(* PLC project Unnamed, Unknown Unnamed 1 *)
(* stored: creationDateTime 2023-05-15T12:31:37, modificationDateTime 2023-06-23T13:12:46 *)

PROGRAM thermal_level_controller
  VAR
    in_valve AT %QX0.0 : BOOL := false;
    out_valve AT %QX0.1 : BOOL := false;
    start_button AT %IX0.0 : BOOL := false;
    low_level AT %IX0.1 : BOOL := false;
    high_level AT %IX0.2 : BOOL := false;
    heater_current AT %QW0 : UINT := 0;
    temperature AT %IW0 : UINT := 0;
  END_VAR
  VAR
    thermal_control_active : BOOL := false;
  END_VAR

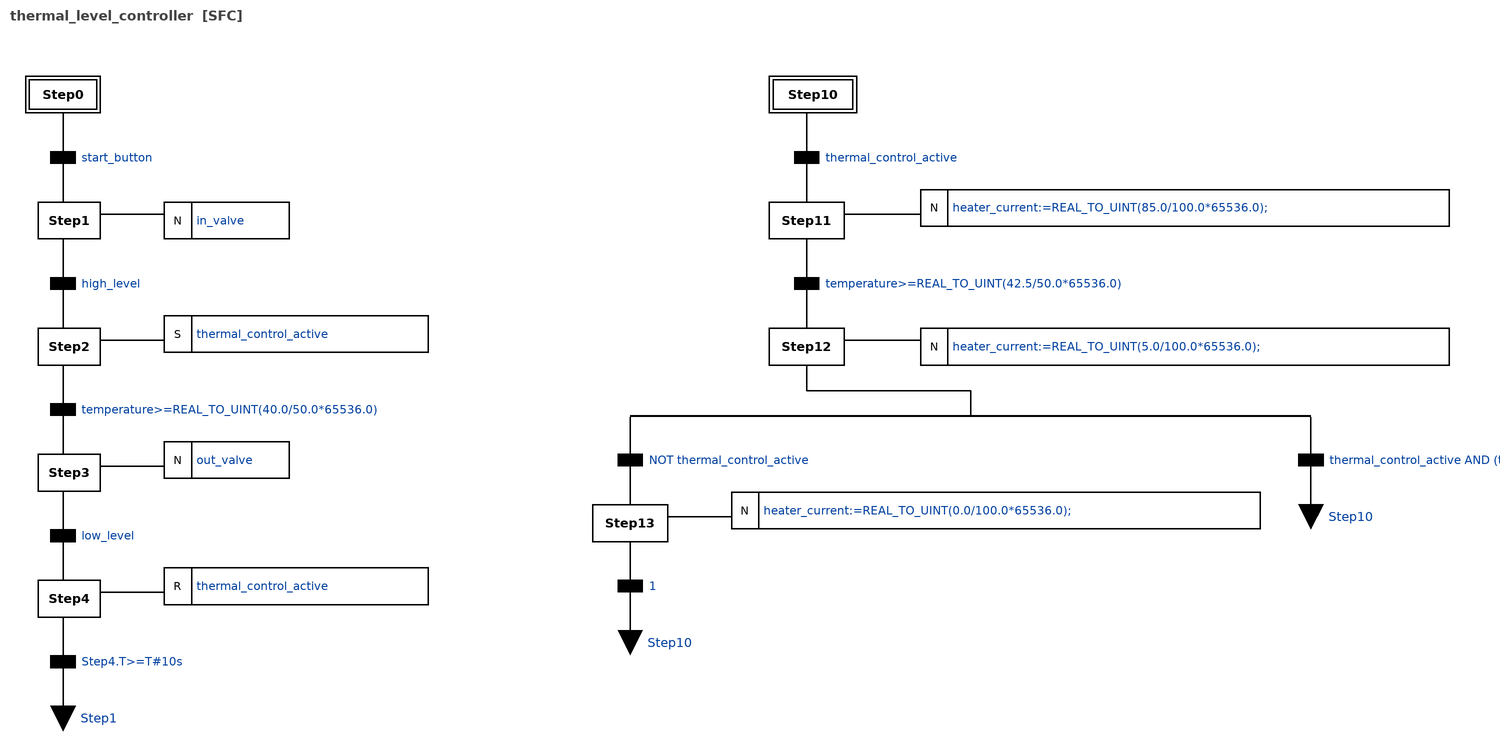
INITIAL_STEP Step0:
END_STEP
TRANSITION FROM Step0 TO Step1
  := start_button;
END_TRANSITION
INITIAL_STEP Step10:
END_STEP
TRANSITION FROM Step10 TO Step11
  := thermal_control_active;
END_TRANSITION
STEP Step1:
  in_valve(N);
END_STEP
TRANSITION FROM Step1 TO Step2
  := high_level;
END_TRANSITION
STEP Step11:
  STEP11_INLINE1(N);
END_STEP
ACTION STEP11_INLINE1:
  heater_current:=REAL_TO_UINT(85.0/100.0*65536.0);
END_ACTION
TRANSITION FROM Step11 TO Step12
  := temperature>=REAL_TO_UINT(42.5/50.0*65536.0);
END_TRANSITION
STEP Step2:
  thermal_control_active(S);
END_STEP
TRANSITION FROM Step2 TO Step3
  := temperature>=REAL_TO_UINT(40.0/50.0*65536.0);
END_TRANSITION
STEP Step12:
  STEP12_INLINE2(N);
END_STEP
ACTION STEP12_INLINE2:
  heater_current:=REAL_TO_UINT(5.0/100.0*65536.0);
END_ACTION
TRANSITION FROM Step12 TO Step10
  := thermal_control_active AND (temperature<=REAL_TO_UINT(37.5/50.0*65536.0));
END_TRANSITION
TRANSITION FROM Step12 TO Step13
  := NOT thermal_control_active;
END_TRANSITION
STEP Step3:
  out_valve(N);
END_STEP
TRANSITION FROM Step3 TO Step4
  := low_level;
END_TRANSITION
STEP Step13:
  STEP13_INLINE3(N);
END_STEP
ACTION STEP13_INLINE3:
  heater_current:=REAL_TO_UINT(0.0/100.0*65536.0);
END_ACTION
TRANSITION FROM Step13 TO Step10
  := 1;
END_TRANSITION
STEP Step4:
  thermal_control_active(R);
END_STEP
TRANSITION FROM Step4 TO Step1
  := Step4.T>=T#10s;
END_TRANSITION
END_PROGRAM

CONFIGURATION Config0
  RESOURCE Res0 ON PLC
    TASK task0(INTERVAL := T#20ms, PRIORITY := 0);
    PROGRAM instance0 WITH task0 : thermal_level_controller;
  END_RESOURCE
END_CONFIGURATION
